PROGRAM MAIN_1MS
VAR
END_VAR

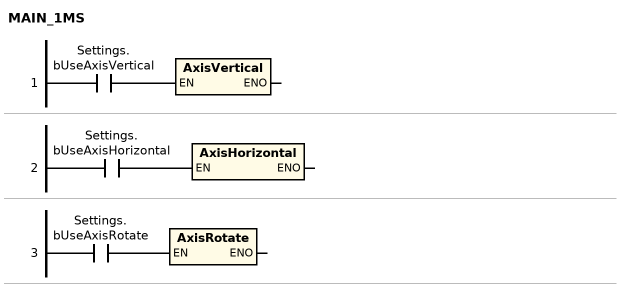
// NETWORK 1
IF Settings.bUseAxisVertical THEN AxisVertical(); END_IF

// NETWORK 2
IF Settings.bUseAxisHorizontal THEN AxisHorizontal(); END_IF

// NETWORK 3
IF Settings.bUseAxisRotate THEN AxisRotate(); END_IF

END_PROGRAM

(* stored: Version 1.1.0.1, ProductVersion 3.1.4024.12
   POU MAIN_1MS: Id {6901df58-f5cb-4ca8-b237-65ad212396c6}, SpecialFunc None *)
